FUNCTION_BLOCK FB_Test_MainFSM EXTENDS TcUnit.FB_TestSuite
VAR
	main_fsm : FB_Main_FSM;
END_VAR

Boot_To_Sync();
Emergency_Command();

METHOD Boot_To_Sync : REFERENCE TO FB_Test
VAR_INPUT
END_VAR
TEST('Boot_To_Sync');

GVL_FSM.can_bus_ok			:= TRUE;
GVL_FSM.safety_inputs_valid	:= TRUE;
GVL_FSM.ethercat_ready		:= TRUE;

main_fsm();

AssertEquals_INT(
	Expected 	:= E_PodState.STATE_SYNC,
	Actual		:= main_fsm.currentState,
	Message		:= 'FSM should transition Boot -> Sync'
);

TEST_FINISHED();
END_METHOD

METHOD Emergency_Command : REFERENCE TO FB_Test
VAR_INPUT
END_VAR
TEST('Emergency_Command');

main_fsm.SetState(newState 	:= E_PodState.STATE_DEMO);
main_fsm.currentCmd		:= E_Command.CMD_EMERGENCY;

main_fsm();

AssertEquals_INT(
	Expected 	:= E_PodState.STATE_EMERGENCY,
	Actual		:= main_fsm.currentState,
	Message		:= 'FSM should transition Boot -> Sync'
);

AssertEquals_BOOL(
	Expected 	:= TRUE,
	Actual		:= main_fsm.criticalFault,
	Message		:= 'FSM should signify the critical state'
);

AssertTrue(
	main_fsm.fb_handle_emergency.busy,
	Message 	:= 'Handle Emergency should be called'
);

TEST_FINISHED();
END_METHOD

END_FUNCTION_BLOCK

(* stored: Version 1.1.0.1
   POU FB_Test_MainFSM: Id {d73df427-cc73-4c5c-8bd4-affee78edae7}, SpecialFunc None
   Method Boot_To_Sync: Id {90e1571a-c972-4c67-8c2c-de9b5672896b}
   Method Emergency_Command: Id {593991bd-eb70-44cf-ac1b-cdf507eb8587} *)
